// TIA Portal V19 program export: 2 tag tables, 0 data types, 0 data blocks, 1 code blocks (in call order from the OBs), 0 instance data blocks

VAR_GLOBAL   // PLC tag table "Default tag table"
   "Conveyor 0" AT %Q0.0 : Bool;
   "memory-eme" AT %M0.0 : Bool;
END_VAR

VAR_GLOBAL   // PLC tag table "Tag table from XML_1"
   "At 1" AT %I0.0 : Bool;
   "At 2" AT %I0.1 : Bool;
   "At 3" AT %I0.2 : Bool;
   "At elevator" AT %I0.3 : Bool;
   "At entry" AT %I0.4 : Bool;
   "At exit" AT %I0.5 : Bool;
   "At 0 (low)" AT %I0.6 : Bool;
   "At 0 (high)" AT %I0.7 : Bool;
   "At 1 (low)" AT %I1.0 : Bool;
   "At 1 (high)" AT %I1.1 : Bool;
   "At 2 (low)" AT %I1.2 : Bool;
   "At 2 (high)" AT %I1.3 : Bool;
   "At 3 (low)" AT %I1.4 : Bool;
   "At 3 (high)" AT %I1.5 : Bool;
   Start AT %I1.6 : Bool;
   Reset AT %I1.7 : Bool;
   Stop AT %I2.0 : Bool;
   "Emergency stop" AT %I2.1 : Bool;
   Auto AT %I2.2 : Bool;
   "Diffuse Sensor 0" AT %I2.3 : Bool;
   "Diffuse Sensor 1" AT %I2.4 : Bool;
   "Diffuse Sensor 2" AT %I2.5 : Bool;
   "Diffuse Sensor 3" AT %I2.6 : Bool;
   "Conveyor 1" AT %Q0.1 : Bool;
   "Conveyor 2" AT %Q0.2 : Bool;
   "Conveyor 3" AT %Q0.3 : Bool;
   "Exit conveyor" AT %Q0.4 : Bool;
   Load AT %Q0.5 : Bool;
   Unload AT %Q0.6 : Bool;
   Up AT %Q0.7 : Bool;
   Down AT %Q1.0 : Bool;
   Slow AT %Q1.1 : Bool;
   "Warning light" AT %Q1.2 : Bool;
   "Start light" AT %Q1.3 : Bool;
   "Reset light" AT %Q1.4 : Bool;
   "Stop light" AT %Q1.5 : Bool;
   "Floor 1" AT %Q1.6 : Bool;
   "Floor 2" AT %Q1.7 : Bool;
   "Floor 3" AT %Q2.0 : Bool;
   "Green 1" AT %Q2.1 : Bool;
   "Yellow 1" AT %Q2.2 : Bool;
   "Red 1" AT %Q2.3 : Bool;
   "Green 2" AT %Q2.4 : Bool;
   "Yellow 2" AT %Q2.5 : Bool;
   "Red 2" AT %Q2.6 : Bool;
   "Green 3" AT %Q2.7 : Bool;
   "Yellow 3" AT %Q3.0 : Bool;
   "Red 3" AT %Q3.1 : Bool;
   Display AT %QD100 : DInt;
END_VAR

ORGANIZATION_BLOCK "Main"   // OB1, LAD, ProgramCycle
TITLE = "Main Program Sweep (Cycle)"
{ S7_Optimized_Access := 'TRUE' }
// stored: SetENOAutomatically false
   VAR_INPUT
      Initial_Call : Bool;   // Initial call of this OB
      Remanence : Bool;   // =True, if remanent data are available
   END_VAR
   VAR_TEMP   // added for the SCL form of the ladder/FBD networks
      _w1 : Bool;
   END_VAR
BEGIN

REGION Network 1
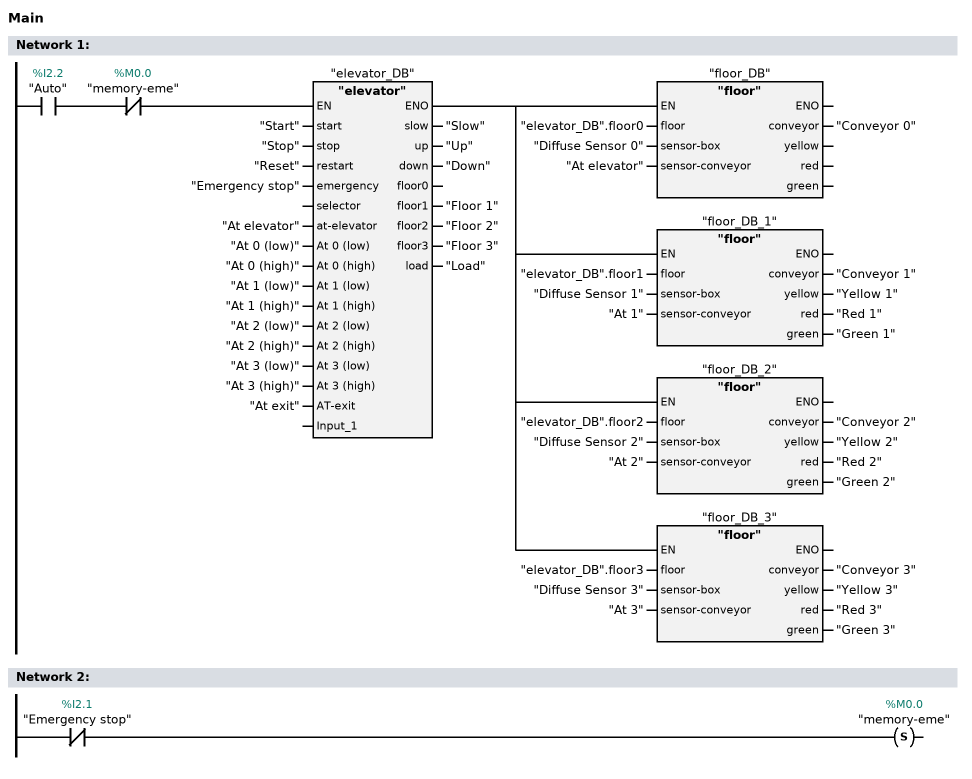
   RUNG wire#powerrail
      Contact( "Auto" )
      I_Contact( "memory-eme" )
      "elevator_DB"(start := "Start", stop := "Stop", restart := "Reset", emergency := "Emergency stop", selector :=, "at-elevator" := "At elevator", "At 0 (low)" := "At 0 (low)", "At 0 (high)" := "At 0 (high)", "At 1 (low)" := "At 1 (low)", "At 1 (high)" := "At 1 (high)", "At 2 (low)" := "At 2 (low)", "At 2 (high)" := "At 2 (high)", "At 3 (low)" := "At 3 (low)", "At 3 (high)" := "At 3 (high)", "AT-exit" := "At exit", Input_1 :=, slow => "Slow", up => "Up", down => "Down", floor0 =>, floor1 => "Floor 1", floor2 => "Floor 2", floor3 => "Floor 3", load => "Load")
      wire#w1
      "floor_DB"(floor := "elevator_DB".floor0, "sensor-box" := "Diffuse Sensor 0", "sensor-conveyor" := "At elevator", conveyor => "Conveyor 0", yellow =>, red =>, green =>)
   END_RUNG
   RUNG wire#w1
      "floor_DB_1"(floor := "elevator_DB".floor1, "sensor-box" := "Diffuse Sensor 1", "sensor-conveyor" := "At 1", conveyor => "Conveyor 1", yellow => "Yellow 1", red => "Red 1", green => "Green 1")
   END_RUNG
   RUNG wire#w1
      "floor_DB_2"(floor := "elevator_DB".floor2, "sensor-box" := "Diffuse Sensor 2", "sensor-conveyor" := "At 2", conveyor => "Conveyor 2", yellow => "Yellow 2", red => "Red 2", green => "Green 2")
   END_RUNG
   RUNG wire#w1
      "floor_DB_3"(floor := "elevator_DB".floor3, "sensor-box" := "Diffuse Sensor 3", "sensor-conveyor" := "At 3", conveyor => "Conveyor 3", yellow => "Yellow 3", red => "Red 3", green => "Green 3")
   END_RUNG
   // the same network as SCL:
   "elevator_DB"(EN := "Auto" AND NOT "memory-eme",   // "elevator"
                 start := "Start",
                 stop := "Stop",
                 restart := "Reset",
                 emergency := "Emergency stop",
                 "at-elevator" := "At elevator",
                 "At 0 (low)" := "At 0 (low)",
                 "At 0 (high)" := "At 0 (high)",
                 "At 1 (low)" := "At 1 (low)",
                 "At 1 (high)" := "At 1 (high)",
                 "At 2 (low)" := "At 2 (low)",
                 "At 2 (high)" := "At 2 (high)",
                 "At 3 (low)" := "At 3 (low)",
                 "At 3 (high)" := "At 3 (high)",
                 "AT-exit" := "At exit",
                 slow => "Slow",
                 up => "Up",
                 down => "Down",
                 floor1 => "Floor 1",
                 floor2 => "Floor 2",
                 floor3 => "Floor 3",
                 load => "Load",
                 ENO => #_w1);
   IF #_w1 THEN
       "floor_DB"(floor := "elevator_DB".floor0,   // "floor"
                  "sensor-box" := "Diffuse Sensor 0",
                  "sensor-conveyor" := "At elevator",
                  conveyor => "Conveyor 0");
       "floor_DB_1"(floor := "elevator_DB".floor1,   // "floor"
                    "sensor-box" := "Diffuse Sensor 1",
                    "sensor-conveyor" := "At 1",
                    conveyor => "Conveyor 1",
                    yellow => "Yellow 1",
                    red => "Red 1",
                    green => "Green 1");
       "floor_DB_2"(floor := "elevator_DB".floor2,   // "floor"
                    "sensor-box" := "Diffuse Sensor 2",
                    "sensor-conveyor" := "At 2",
                    conveyor => "Conveyor 2",
                    yellow => "Yellow 2",
                    red => "Red 2",
                    green => "Green 2");
       "floor_DB_3"(floor := "elevator_DB".floor3,   // "floor"
                    "sensor-box" := "Diffuse Sensor 3",
                    "sensor-conveyor" := "At 3",
                    conveyor => "Conveyor 3",
                    yellow => "Yellow 3",
                    red => "Red 3",
                    green => "Green 3");
   END_IF;
END_REGION

REGION Network 2
   RUNG wire#powerrail
      I_Contact( "Emergency stop" )
      S_Coil( "memory-eme" )
   END_RUNG
   // the same network as SCL:
   IF NOT "Emergency stop" THEN "memory-eme" := TRUE; END_IF;
END_REGION
END_ORGANIZATION_BLOCK
